RoboDK station: Stringer B-Corner-Bot-Long-BOX2.rdk

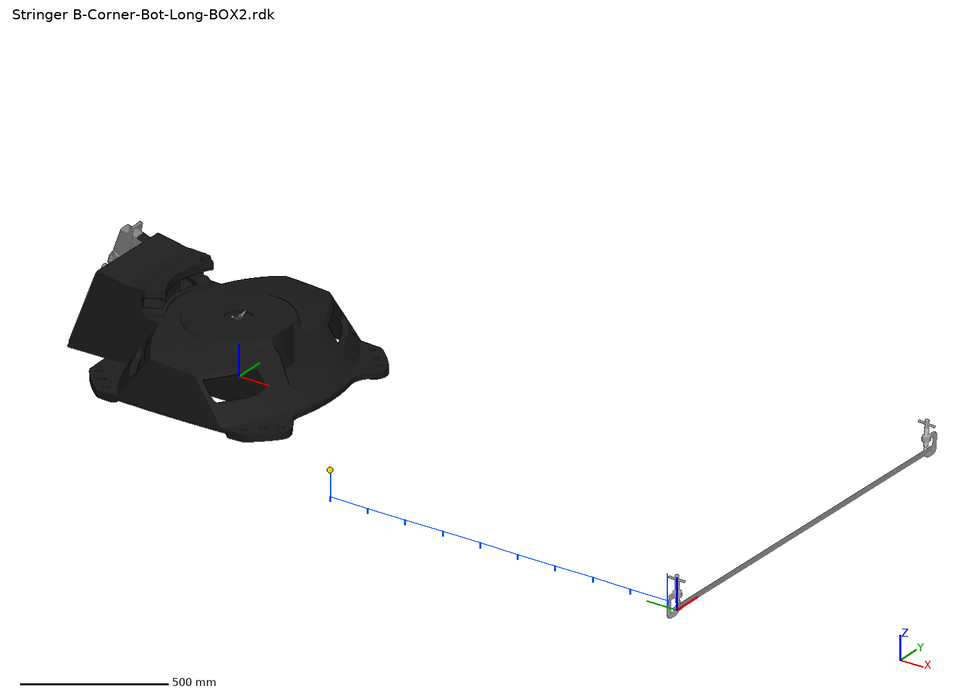
[picture v0: the station drawn from its stored meshes, robots at their saved joint values, targets as dots, program paths as lines]
Station Stringer B-Corner-Bot-Long-BOX2 (saved by RoboDK 5.2.3). Poses are relative to the parent item; angles as X-Y-Z fixed-axis rotations.
  - frame KUKA KR 210 R2700 extra Base at (0, 0, 0) mm
    - robot KUKA KR 210 R2700 extra: 6 axes, payload 210 kg, reach 2696 mm, repeatability 0.06 mm, weight 1068 kg
        joint limits [-185, -140, -120, -350, -125, -350] to [185, -5, 155, 350, 125, 350]; home [0, -90, 90, 0, 0, 0]; saved at [-1.792, -34.007, 111.814, 177.5, 26.815, -179.161]
      - tool Spindle, TCP at (32, 0, 260) mm, rotated rx 0 ry 39 rz 0 deg, size 157.3 x 72 x 259.9 mm
  - frame Frame 2 at (1800, 0, -372.68) mm, rotated rx 0 ry 0 rz 90 deg
    - object Stringer B-Corner-Bot-Long-BOX2 at (0, 22.5, 0) mm, rotated rx 0 ry 0 rz -90 deg, 10 curves, geometry from Point 10
    - object L-Stringer B-corner-bottom-long - box2 at (0, 0, 0) mm, size 1499.5 x 20 x 20 mm, geometry from L-Stringer B-corner-bottom-long - box2.stl
  - machining project Point settings: rotZ(0) | rotX(0)*rotY(0) | rotz(0) | onStart | onPathStart | onApproach | onPoint | onRetract | onFinish | SetRPM(%1) | SetTool(%1) | Extruder(%1) | default | default | OutOnMov(%1) | OutOffMov(%1) | onPathFinish | M_RunCode(%1)
  - program Point (61 instructions, listed below)
  - object FinalClamp at (1784.91, 22.27, -312.83) mm, rotated rx -178.1 ry 87.86 rz 0 deg, size 145.3 x 71.1 x 72 mm, geometry from FinalClamp.stp
  - object FinalClamp2 at (1788.86, 1477.69, -310.22) mm, rotated rx 180 ry 87.26 rz 180 deg, size 145.3 x 71.1 x 72 mm, geometry from FinalClamp.stp
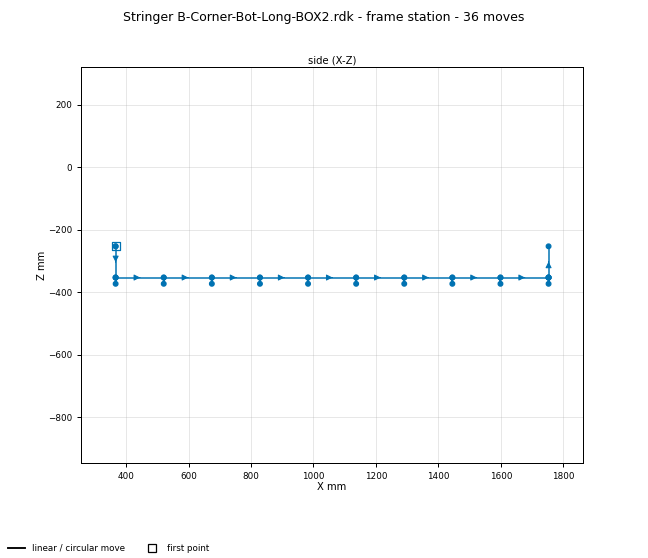
[picture p0: tool path of Stringer B-Corner-Bot-Long-BOX2.rdk in frame station, 36 of 36 moves have a stored position in this frame; points joined in program order, loops and branches not executed]

--- program Point (robot KUKA KR 210 R2700 extra) ---
  Smooth(1)
  Set speed (1000.0 mm/s)
  Set Ref.: Frame 2
  Set Tool: Spindle
  Show Spindle
  MoveJ 1 to (12.5, 1433.43, 120) mm, rotated rx -180 ry 0 rz -180 deg; joints [-43.398, -23.142, 76.755, 77.872, 26.247, -112.836]
  MoveL 2 to (12.5, 1433.43, 120) mm, rotated rx -180 ry 0 rz -180 deg; joints [-43.398, -23.142, 76.755, 77.872, 26.247, -112.836]
  MoveL 3 to (12.5, 1433.43, 20) mm, rotated rx 180 ry 0 rz 180 deg; joints [-43.398, -18.887, 74.254, 81.395, 25.932, -116.758]
  MoveL 4 to (12.5, 1433.43, 20) mm, rotated rx 180 ry 0 rz 180 deg; joints [-43.398, -18.887, 74.254, 81.395, 25.932, -116.758]
  Set speed (50.0 mm/s)
  MoveL 5 to (12.5, 1433.43, 0) mm, rotated rx 180 ry 0 rz 180 deg; joints [-43.398, -18.021, 73.699, 82.029, 25.887, -117.464]
  MoveL 6 to (12.5, 1433.43, 20) mm, rotated rx 180 ry 0 rz 180 deg; joints [-43.398, -18.887, 74.254, 81.395, 25.932, -116.758]
  Set speed (1000.0 mm/s)
  MoveL 7 to (12.5, 1279.43, 20) mm, rotated rx 180 ry 0 rz -180 deg; joints [-40.164, -21.512, 81.55, 94.02, 24.01, -127.66]
  Set speed (50.0 mm/s)
  MoveL 8 to (12.5, 1279.43, 0) mm, rotated rx -180 ry 0 rz -180 deg; joints [-40.164, -20.625, 81.008, 94.793, 24.037, -128.506]
  MoveL 9 to (12.5, 1279.43, 20) mm, rotated rx 180 ry 0 rz -180 deg; joints [-40.164, -21.512, 81.55, 94.02, 24.01, -127.66]
  Set speed (1000.0 mm/s)
  MoveL 10 to (12.5, 1125.43, 20) mm, rotated rx -180 ry 0 rz -180 deg; joints [-36.59, -23.597, 87.858, 107.415, 23.151, -138.82]
  Set speed (50.0 mm/s)
  MoveL 11 to (12.5, 1125.43, 0) mm, rotated rx -180 ry 0 rz -180 deg; joints [-36.59, -22.684, 87.32, 108.248, 23.266, -139.726]
  MoveL 12 to (12.5, 1125.43, 20) mm, rotated rx -180 ry 0 rz -180 deg; joints [-36.59, -23.597, 87.858, 107.415, 23.151, -138.82]
  Set speed (1000.0 mm/s)
  MoveL 13 to (12.5, 971.43, 20) mm, rotated rx -180 ry 0 rz -180 deg; joints [-32.652, -25.224, 93.294, 120.659, 23.248, -149.302]
  Set speed (50.0 mm/s)
  MoveL 14 to (12.5, 971.43, 0) mm, rotated rx 180 ry 0 rz 180 deg; joints [-32.652, -24.283, 92.753, 121.455, 23.455, -150.169]
  MoveL 15 to (12.5, 971.43, 20) mm, rotated rx -180 ry 0 rz -180 deg; joints [-32.652, -25.224, 93.294, 120.659, 23.248, -149.302]
  Set speed (1000.0 mm/s)
  MoveL 16 to (12.5, 817.43, 20) mm, rotated rx 180 ry 0 rz -180 deg; joints [-28.335, -26.457, 97.915, 132.95, 24.084, -158.293]
  Set speed (50.0 mm/s)
  MoveL 17 to (12.5, 817.43, 0) mm, rotated rx -180 ry 0 rz -180 deg; joints [-28.335, -25.487, 97.369, 133.635, 24.374, -159.045]
  MoveL 18 to (12.5, 817.43, 20) mm, rotated rx 180 ry 0 rz -180 deg; joints [-28.335, -26.457, 97.915, 132.95, 24.084, -158.293]
  Set speed (1000.0 mm/s)
  MoveL 19 to (12.5, 663.43, 20) mm, rotated rx 180 ry 0 rz 180 deg; joints [-23.636, -27.353, 101.747, 143.916, 25.365, -165.418]
  Set speed (50.0 mm/s)
  MoveL 20 to (12.5, 663.43, 0) mm, rotated rx 180 ry 0 rz 180 deg; joints [-23.636, -26.357, 101.194, 144.459, 25.725, -166.019]
  MoveL 21 to (12.5, 663.43, 20) mm, rotated rx 180 ry 0 rz 180 deg; joints [-23.636, -27.353, 101.747, 143.916, 25.365, -165.418]
  Set speed (1000.0 mm/s)
  MoveL 22 to (12.5, 509.43, 20) mm, rotated rx 180 ry 0 rz 180 deg; joints [-18.575, -27.97, 104.796, 153.593, 26.792, -170.731]
  Set speed (50.0 mm/s)
  MoveL 23 to (12.5, 509.43, 0) mm, rotated rx 180 ry 0 rz 180 deg; joints [-18.575, -26.95, 104.235, 153.991, 27.203, -171.178]
  MoveL 24 to (12.5, 509.43, 20) mm, rotated rx 180 ry 0 rz 180 deg; joints [-18.575, -27.97, 104.796, 153.593, 26.792, -170.731]
  Set speed (1000.0 mm/s)
  MoveL 25 to (12.5, 355.43, 20) mm, rotated rx 180 ry 0 rz 180 deg; joints [-13.195, -28.365, 107.055, 162.236, 28.09, -174.545]
  Set speed (50.0 mm/s)
  MoveL 26 to (12.5, 355.43, 0) mm, rotated rx -180 ry 0 rz -180 deg; joints [-13.195, -27.326, 106.487, 162.501, 28.539, -174.845]
  MoveL 27 to (12.5, 355.43, 20) mm, rotated rx 180 ry 0 rz 180 deg; joints [-13.195, -28.365, 107.055, 162.236, 28.09, -174.545]
  Set speed (1000.0 mm/s)
  MoveL 28 to (12.5, 201.43, 20) mm, rotated rx -180 ry 0 rz -180 deg; joints [-7.569, -28.588, 108.517, 170.169, 29.043, -177.281]
  Set speed (50.0 mm/s)
  MoveL 29 to (12.5, 201.43, 0) mm, rotated rx 180 ry 0 rz -180 deg; joints [-7.569, -27.536, 107.944, 170.313, 29.514, -177.446]
  MoveL 30 to (12.5, 201.43, 20) mm, rotated rx -180 ry 0 rz -180 deg; joints [-7.569, -28.588, 108.517, 170.169, 29.043, -177.281]
  Set speed (1000.0 mm/s)
  MoveL 31 to (12.5, 47.43, 20) mm, rotated rx 180 ry 0 rz -180 deg; joints [-1.792, -28.679, 109.172, 177.709, 29.499, -179.399]
  Set speed (50.0 mm/s)
  MoveL 32 to (12.5, 47.43, 0) mm, rotated rx 180 ry 0 rz 180 deg; joints [-1.792, -27.622, 108.596, 177.743, 29.98, -179.438]
  MoveL 33 to (12.5, 47.43, 20) mm, rotated rx 180 ry 0 rz -180 deg; joints [-1.792, -28.679, 109.172, 177.709, 29.499, -179.399]
  MoveL 34 to (12.5, 47.43, 20) mm, rotated rx 180 ry 0 rz -180 deg; joints [-1.792, -28.679, 109.172, 177.709, 29.499, -179.399]
  Set speed (1000.0 mm/s)
  MoveL 35 to (12.5, 47.43, 20) mm, rotated rx 180 ry 0 rz -180 deg; joints [-1.792, -28.679, 109.172, 177.709, 29.499, -179.399]
  MoveL 36 to (12.5, 47.43, 120) mm, rotated rx 180 ry 0 rz -180 deg; joints [-1.792, -34.007, 111.814, 177.5, 26.815, -179.161]
